FUNCTION_BLOCK FB_SaMElementCompleting EXTENDS FB_SaMElement
VAR
END_VAR

METHOD FB_init : BOOL
VAR_INPUT
	bInitRetains : BOOL; // if TRUE, the retain variables are initialized (warm start / cold start)
	bInCopyCode : BOOL;  // if TRUE, the instance afterwards gets moved into the copy code (online change)
END_VAR
THIS^.bTypeActive		:= TRUE;

THIS^.SetText (eLocation := E_BaseLocation.pl, wsDescription := "Kompletowanie");
THIS^.SetText (eLocation := E_BaseLocation.en, wsDescription := "Completing");
THIS^.SetText (eLocation := E_BaseLocation.de, wsDescription := "Abschluss");
THIS^.SetName (stName := THIS^.GetTexts ());
END_METHOD

METHOD public GetNextState : E_BaseMachineState
VAR_INPUT
END_VAR
GetNextState		:= E_BaseMachineState.Complete;
END_METHOD

METHOD PUBLIC InvokeStateForTopElement : BOOL
VAR_INPUT
	itfTopElement		: ITF_BaseSaMStateMethod;
END_VAR
InvokeStateForTopElement	:= itfTopElement.SP_Completing ();
END_METHOD

END_FUNCTION_BLOCK

(* stored: Version 1.1.0.1
   POU FB_SaMElementCompleting: Id {95f25625-e0e4-0748-3f6e-13f41076680a}, SpecialFunc None
   Method FB_init: Id {28071300-25d2-03c8-3942-b78a77afb5f4}
   Method GetNextState: Id {c039c46f-2bb2-047c-3f3c-f89a9ffebbab}
   Method InvokeStateForTopElement: Id {95335b1f-6c20-03bf-2e42-43f816aa825b} *)
